// TIA Portal V16 export
// export: Created 2021-04-13T11:10:14.4344979Z, ExportSetting WithDefaults, DisplayName Totally Integrated Automation Portal, DisplayVersion V16, DisplayName TIA Portal Version Control Interface, DisplayVersion V16, DisplayName TIA Portal Openness, DisplayVersion V16, DisplayName STEP 7 Professional, DisplayVersion V16, DisplayName STEP 7 Safety, DisplayVersion V16, DisplayName WinCC Unified SCADA Engineering System, DisplayVersion V16
FUNCTION_BLOCK "modbus_SenecaConnectPort2"   // FB14, LAD
{ S7_Optimized_Access := 'TRUE' }
VERSION : 0.1
// stored: AutoNumber false, IsIECCheckEnabled false, IsRetainMemResEnabled false, MemoryReserve 100, SetENOAutomatically false, UDAEnableTagReadback false
   VAR_INPUT
      port : PORT;   // порт для подключения
      arrayAddressModbus : Array[0..12] of UInt;
      Offset_array_bits : SInt;
   END_VAR
   VAR_IN_OUT
      calibrateZero : Array[0..12] of Bool;
      taraZero : Array[0..12] of Bool;
      currentWeight : Array[0..12] of Real;
   END_VAR
   VAR
      MB_COMM_LOAD : MB_COMM_LOAD;
      MB_MASTER : MB_MASTER;
      Data_toMB_MASTER : Struct
         REQ : Bool;
         MB_ADDR : UInt;
         MODE : USInt;
         DATA_ADDR : UDInt;
         DATA_LEN : UInt;
         DONE : Bool;
         BUSY : Bool;
         ERROR : Bool;
      END_STRUCT;
      Seneca : Struct
         TON_changeStep : TON_TIME;
         TON_Start { S7_SetPoint := 'True'} : Bool;
         "Step" : SInt;
      END_STRUCT;
      tmpWeight : Array[0..12] of DWord;
      restartPort : Bool;   // перезагрузка Modbus
      needCalibrate : Bool;   // проверка на необходимость калибровки или тарирования
      testDone : Struct
         ton1 : TON_TIME;
         pulse_High : Bool;
         ton2 : TON_TIME;
         p_trig : Bool;
         ctu1 : CTU_INT;
      END_STRUCT;
   END_VAR
   VAR_TEMP
      index : DInt;
      tmpIndex : DInt;
      i : DInt;
   END_VAR
   // MB_COMM_LOAD.RETRIES := 1;
   VAR_TEMP   // added for the SCL form of the ladder/FBD networks
      _w1 : Bool;
   END_VAR
BEGIN

REGION Network 1: ИНИЦИАЛИЗИРУЕМ ПОРТ
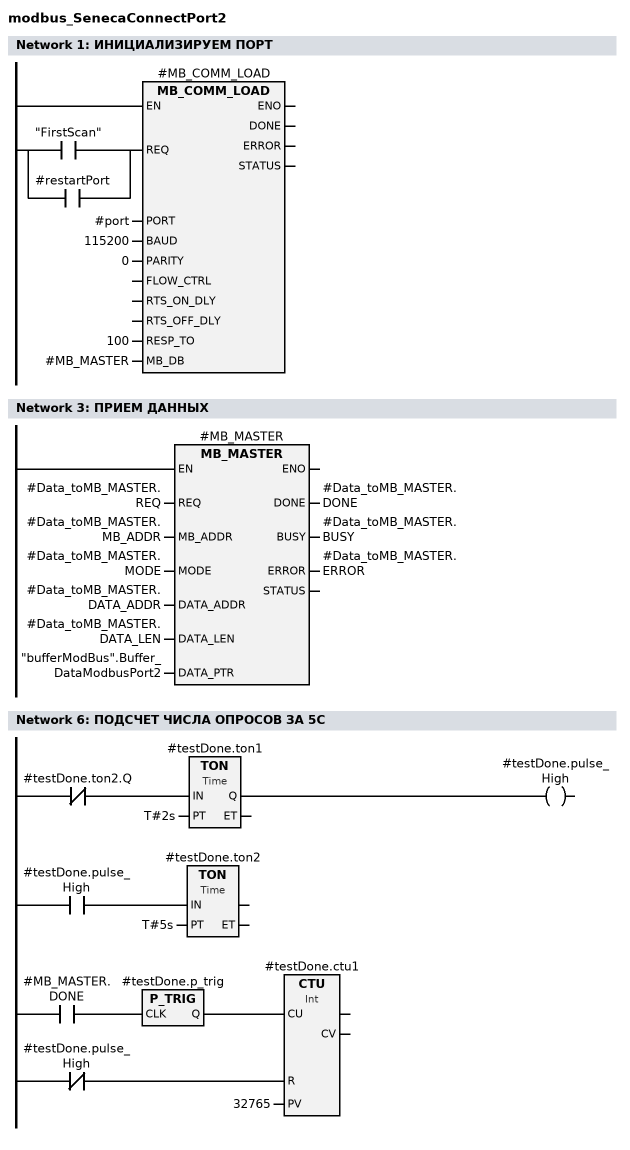
   RUNG wire#powerrail
      #MB_COMM_LOAD.MB_COMM_LOAD(REQ := wire#w1, PORT := #port, BAUD := 115200, PARITY := 0, FLOW_CTRL :=, RTS_ON_DLY :=, RTS_OFF_DLY :=, RESP_TO := 100, MB_DB := #MB_MASTER, DONE =>, ERROR =>, STATUS =>)
   END_RUNG
   RUNG wire#powerrail
      Contact( "FirstScan" )
   END_RUNG wire#w1
   RUNG wire#powerrail
      Contact( #restartPort )
   END_RUNG wire#w1
   // the same network as SCL:
   #MB_COMM_LOAD(REQ := "FirstScan" OR #restartPort,   // MB_COMM_LOAD
                 PORT := #port,
                 BAUD := 115200,
                 PARITY := 0,
                 RESP_TO := 100,
                 MB_DB := #MB_MASTER);
END_REGION

REGION Network 2 (SCL): ОБМЕН
   #Seneca.TON_changeStep(IN := #Seneca.TON_Start,
                          PT := t#50ms);

   CASE #Seneca.Step OF

       1: //ЧИТАЕМ ЗНАЧЕНИЕ ВЕСА С ПЕРВОГО МОДУЛЯ

           #index := 1 + #Offset_array_bits;//заполнять функцию будем через индекс чтобы меньше писать
           "rcvDataWeight"(ADDR_DEVICE := #arrayAddressModbus[#index],
                           Ton_changeStep := #Seneca.TON_changeStep.Q,
                           Ton_Start := #Seneca.TON_Start,
                           "Step" := #Seneca.Step,
                           MB_MASTER := #Data_toMB_MASTER);

       2://ЧИТАЕМ ЗНАЧЕНИЕ ВЕСА СО ВТОРОГО МОДУЛЯ
           #index := 2 + #Offset_array_bits;//заполнять функцию будем через индекс чтобы меньше писать
           "rcvDataWeight"(ADDR_DEVICE := #arrayAddressModbus[#index],
                           Ton_changeStep := #Seneca.TON_changeStep.Q,
                           Ton_Start := #Seneca.TON_Start,
                           "Step" := #Seneca.Step,
                           MB_MASTER := #Data_toMB_MASTER);

       7: // КАЛИБРОВКА 0 ДЛЯ ПЕРВОГО МОДУЛЯ и ТАРИРОВАНИЕ
           #i := 0;
           FOR #i := 1 TO 6 DO
               IF #calibrateZero[#i + #Offset_array_bits] OR #taraZero[#i + #Offset_array_bits] THEN
                   #needCalibrate := true;
                   EXIT;
               END_IF;
           END_FOR;

           IF #needCalibrate THEN
               #index := 1 + #Offset_array_bits;//заполнять функцию будем через индекс чтобы меньше писать
               IF #calibrateZero[#index] OR #taraZero[#index] THEN
                   "sndCALIBR&Tara"(ADDR_DEVICE := #arrayAddressModbus[#index],
                                    ton_changeStep := #Seneca.TON_changeStep.Q,
                                    MB_MASTER := #Data_toMB_MASTER,
                                    Ton_Start := #Seneca.TON_Start,
                                    Calibrate := #calibrateZero[#index],
                                    Buffer := "bufferModBus".Buffer_DataModbusPort2,
                                    "Step" := #Seneca.Step,
                                    Tara := #taraZero[#index]);
               ELSE
                   #Seneca.Step := #Seneca.Step + 1;
               END_IF;
           ELSE
               #Seneca.Step := 1;
           END_IF;

       8:// КАЛИБРОВКА 0 ДЛЯ ВТОРОГО МОДУЛЯ и ТАРИРОВАНИЕ
           #index := 2 + #Offset_array_bits;//заполнять функцию будем через индекс чтобы меньше писать
           IF #calibrateZero[#index] OR #taraZero[#index] THEN
               "sndCALIBR&Tara"(ADDR_DEVICE := #arrayAddressModbus[#index],
                                ton_changeStep := #Seneca.TON_changeStep.Q,
                                MB_MASTER := #Data_toMB_MASTER,
                                Ton_Start := #Seneca.TON_Start,
                                Calibrate := #calibrateZero[#index],
                                Buffer := "bufferModBus".Buffer_DataModbusPort2,
                                "Step" := #Seneca.Step,
                                Tara := #taraZero[#index]);
           ELSE
               #Seneca.Step := #Seneca.Step + 1;
           END_IF;

           //////////////////////////////////////////////////////////////////////////////////
           //////////////////////////////////////////////////////////////////////////////////
           //////////////////////////////////////////////////////////////////////////////////
           //////////////////////////////////////////////////////////////////////////////////
       3: //ЧИТАЕМ ЗНАЧЕНИЕ ВЕСА С ТРЕТЬЕГО МОДУЛЯ

           #index := 3 + #Offset_array_bits;//заполнять функцию будем через индекс чтобы меньше писать
           "rcvDataWeight"(ADDR_DEVICE := #arrayAddressModbus[#index],
                           Ton_changeStep := #Seneca.TON_changeStep.Q,
                           Ton_Start := #Seneca.TON_Start,
                           "Step" := #Seneca.Step,
                           MB_MASTER := #Data_toMB_MASTER);

       4://ЧИТАЕМ ЗНАЧЕНИЕ ВЕСА С ЧЕТВЕРТОГО МОДУЛЯ
           #index := 4 + #Offset_array_bits;//заполнять функцию будем через индекс чтобы меньше писать
           "rcvDataWeight"(ADDR_DEVICE := #arrayAddressModbus[#index],
                           Ton_changeStep := #Seneca.TON_changeStep.Q,
                           Ton_Start := #Seneca.TON_Start,
                           "Step" := #Seneca.Step,
                           MB_MASTER := #Data_toMB_MASTER);

       9:// КАЛИБРОВКА 0 ДЛЯ ТРЕТЬЕГО  МОДУЛЯ

           #index := 3 + #Offset_array_bits;//заполнять функцию будем через индекс чтобы меньше писать
           IF #calibrateZero[#index] OR #taraZero[#index] THEN
               "sndCALIBR&Tara"(ADDR_DEVICE := #arrayAddressModbus[#index],
                                ton_changeStep := #Seneca.TON_changeStep.Q,
                                MB_MASTER := #Data_toMB_MASTER,
                                Ton_Start := #Seneca.TON_Start,
                                Calibrate := #calibrateZero[#index],
                                Buffer := "bufferModBus".Buffer_DataModbusPort2,
                                "Step" := #Seneca.Step,
                                Tara := #taraZero[#index]);
           ELSE
               #Seneca.Step := #Seneca.Step + 1;
           END_IF;

       10://КАЛИБРОВКА 0 ДЛЯ ЧЕТВЕРТОГО МОДУЛЯ

           #index := 4 + #Offset_array_bits;//заполнять функцию будем через индекс чтобы меньше писать
           IF #calibrateZero[#index] OR #taraZero[#index] THEN
               "sndCALIBR&Tara"(ADDR_DEVICE := #arrayAddressModbus[#index],
                                ton_changeStep := #Seneca.TON_changeStep.Q,
                                MB_MASTER := #Data_toMB_MASTER,
                                Ton_Start := #Seneca.TON_Start,
                                Calibrate := #calibrateZero[#index],
                                Buffer := "bufferModBus".Buffer_DataModbusPort2,
                                "Step" := #Seneca.Step,
                                Tara := #taraZero[#index]);
           ELSE
               #Seneca.Step := #Seneca.Step + 1;
           END_IF;

           /////////////////////////////////////////////////////////////////////////////////
           ////////////////////////////////////////////////////////////////////////////////
           ////////////////////////////////////////////////////////////////////////////////
           ////////////////////////////////////////////////////////////////////////////////
       5: //ЧИТАЕМ ЗНАЧЕНИЕ ВЕСА С ПЯТОГО МОДУЛЯ
           #index := 5 + #Offset_array_bits;//заполнять функцию будем через индекс чтобы меньше писать
           "rcvDataWeight"(ADDR_DEVICE := #arrayAddressModbus[#index],
                           Ton_changeStep := #Seneca.TON_changeStep.Q,
                           Ton_Start := #Seneca.TON_Start,
                           "Step" := #Seneca.Step,
                           MB_MASTER := #Data_toMB_MASTER);

       6://ЧИТАЕМ ЗНАЧЕНИЕ ВЕСА С ШЕСТОГО МОДУЛЯ
           #index := 6 + #Offset_array_bits;//заполнять функцию будем через индекс чтобы меньше писать
           "rcvDataWeight"(ADDR_DEVICE := #arrayAddressModbus[#index],
                           Ton_changeStep := #Seneca.TON_changeStep.Q,
                           Ton_Start := #Seneca.TON_Start,
                           "Step" := #Seneca.Step,
                           MB_MASTER := #Data_toMB_MASTER);

       11:// КАЛИБРОВКА 0 ДЛЯ ПЯТОГО  МОДУЛЯ

           #index := 5 + #Offset_array_bits;//заполнять функцию будем через индекс чтобы меньше писать
           IF #calibrateZero[#index] OR #taraZero[#index] THEN
               "sndCALIBR&Tara"(ADDR_DEVICE := #arrayAddressModbus[#index],
                                ton_changeStep := #Seneca.TON_changeStep.Q,
                                MB_MASTER := #Data_toMB_MASTER,
                                Ton_Start := #Seneca.TON_Start,
                                Calibrate := #calibrateZero[#index],
                                Buffer := "bufferModBus".Buffer_DataModbusPort2,
                                "Step" := #Seneca.Step,
                                Tara := #taraZero[#index]);
           ELSE
               #Seneca.Step := #Seneca.Step + 1;
           END_IF;

       12:// КАЛИБРОВКА 0 ДЛЯ ШЕСТОГО МОДУЛЯ
           #index := 6 + #Offset_array_bits;//заполнять функцию будем через индекс чтобы меньше писать
           IF #calibrateZero[#index] OR #taraZero[#index] THEN
               "sndCALIBR&Tara"(ADDR_DEVICE := #arrayAddressModbus[#index],
                                ton_changeStep := #Seneca.TON_changeStep.Q,
                                MB_MASTER := #Data_toMB_MASTER,
                                Ton_Start := #Seneca.TON_Start,
                                Calibrate := #calibrateZero[#index],                            Buffer := "bufferModBus".Buffer_DataModbusPort2,
                                "Step" := #Seneca.Step,
                                Tara := #taraZero[#index]);
           ELSE
               #Seneca.Step := #Seneca.Step + 1;
           END_IF;
           #needCalibrate := false;
       ELSE
           #Seneca.Step := 1;
   END_CASE;
END_REGION

REGION Network 3: ПРИЕМ ДАННЫХ
   RUNG wire#powerrail
      #MB_MASTER.MB_MASTER(REQ := #Data_toMB_MASTER.REQ, MB_ADDR := #Data_toMB_MASTER.MB_ADDR, MODE := #Data_toMB_MASTER.MODE, DATA_ADDR := #Data_toMB_MASTER.DATA_ADDR, DATA_LEN := #Data_toMB_MASTER.DATA_LEN, DATA_PTR := "bufferModBus".Buffer_DataModbusPort2, DONE => #Data_toMB_MASTER.DONE, BUSY => #Data_toMB_MASTER.BUSY, ERROR => #Data_toMB_MASTER.ERROR, STATUS =>)
   END_RUNG
   // the same network as SCL:
   #MB_MASTER(REQ := #Data_toMB_MASTER.REQ,   // MB_MASTER
              MB_ADDR := #Data_toMB_MASTER.MB_ADDR,
              MODE := #Data_toMB_MASTER.MODE,
              DATA_ADDR := #Data_toMB_MASTER.DATA_ADDR,
              DATA_LEN := #Data_toMB_MASTER.DATA_LEN,
              DATA_PTR := "bufferModBus".Buffer_DataModbusPort2,
              DONE => #Data_toMB_MASTER.DONE,
              BUSY => #Data_toMB_MASTER.BUSY,
              ERROR => #Data_toMB_MASTER.ERROR);
END_REGION

REGION Network 4 (SCL): Авария опроса модуля
   #index := 0;
   CASE #Seneca.Step OF
       1,7:
           #index := 7;
       2,8:
           #index := 8;
       3,9:
           #index := 9;
       4,10:
           #index := 10;
       5,11:
           #index := 11;
       6,12:
           #index := 12;

   END_CASE;
   IF #Data_toMB_MASTER.ERROR THEN
       "hmi".alarmTest.bit[#index] := true;
   ELSIF #Data_toMB_MASTER.DONE THEN
       "hmi".alarmTest.bit[#index] := FALSE;
   END_IF;
END_REGION

REGION Network 5 (SCL)
   IF #Seneca.Step = 1 AND #Data_toMB_MASTER.DONE THEN
       #tmpIndex := 1 + #Offset_array_bits;
       #tmpWeight[#tmpIndex].%W0 := "bufferModBus".Buffer_DataModbusPort2[1];
       #tmpWeight[#tmpIndex].%W1 := "bufferModBus".Buffer_DataModbusPort2[0];
       #currentWeight[#tmpIndex] := DWORD_TO_REAL(#tmpWeight[#tmpIndex]);
       "bufferModBus".Buffer_DataModbusPort2[0] := 0;
       "bufferModBus".Buffer_DataModbusPort2[1] := 0;

   END_IF;

   IF #Seneca.Step = 2 AND #Data_toMB_MASTER.DONE THEN
       #tmpIndex := 2 + #Offset_array_bits;
       #tmpWeight[#tmpIndex].%W0 := "bufferModBus".Buffer_DataModbusPort2[1];
       #tmpWeight[#tmpIndex].%W1 := "bufferModBus".Buffer_DataModbusPort2[0];
       #currentWeight[#tmpIndex] := DWORD_TO_REAL(#tmpWeight[#tmpIndex]);
       "bufferModBus".Buffer_DataModbusPort2[0] := 0;
       "bufferModBus".Buffer_DataModbusPort2[1] := 0;
   END_IF;

   IF #Seneca.Step = 3 AND #Data_toMB_MASTER.DONE THEN
       #tmpIndex := 3 + #Offset_array_bits;
       #tmpWeight[#tmpIndex].%W0 := "bufferModBus".Buffer_DataModbusPort2[1];
       #tmpWeight[#tmpIndex].%W1 := "bufferModBus".Buffer_DataModbusPort2[0];
       #currentWeight[#tmpIndex] := DWORD_TO_REAL(#tmpWeight[#tmpIndex]);
       "bufferModBus".Buffer_DataModbusPort2[0] := 0;
       "bufferModBus".Buffer_DataModbusPort2[1] := 0;
   END_IF;

   IF #Seneca.Step = 4 AND #Data_toMB_MASTER.DONE THEN
       #tmpIndex := 4 + #Offset_array_bits;
       #tmpWeight[#tmpIndex].%W0 := "bufferModBus".Buffer_DataModbusPort2[1];
       #tmpWeight[#tmpIndex].%W1 := "bufferModBus".Buffer_DataModbusPort2[0];
       #currentWeight[#tmpIndex] := DWORD_TO_REAL(#tmpWeight[#tmpIndex]);
       "bufferModBus".Buffer_DataModbusPort2[0] := 0;
       "bufferModBus".Buffer_DataModbusPort2[1] := 0;
   END_IF;

   IF #Seneca.Step = 5 AND #Data_toMB_MASTER.DONE THEN
       #tmpIndex := 5 + #Offset_array_bits;
       #tmpWeight[#tmpIndex].%W0 := "bufferModBus".Buffer_DataModbusPort2[1];
       #tmpWeight[#tmpIndex].%W1 := "bufferModBus".Buffer_DataModbusPort2[0];
       #currentWeight[#tmpIndex] := DWORD_TO_REAL(#tmpWeight[#tmpIndex]);
       "bufferModBus".Buffer_DataModbusPort2[0] := 0;
       "bufferModBus".Buffer_DataModbusPort2[1] := 0;
   END_IF;

   IF #Seneca.Step = 6 AND #Data_toMB_MASTER.DONE THEN
       #tmpIndex := 6 + #Offset_array_bits;
       #tmpWeight[#tmpIndex].%W0 := "bufferModBus".Buffer_DataModbusPort2[1];
       #tmpWeight[#tmpIndex].%W1 := "bufferModBus".Buffer_DataModbusPort2[0];
       #currentWeight[#tmpIndex] := DWORD_TO_REAL(#tmpWeight[#tmpIndex]);
       "bufferModBus".Buffer_DataModbusPort2[0] := 0;
       "bufferModBus".Buffer_DataModbusPort2[1] := 0;
   END_IF;
END_REGION

REGION Network 6: ПОДСЧЕТ ЧИСЛА ОПРОСОВ ЗА 5С
   RUNG wire#powerrail
      I_Contact( #testDone.ton2.Q )
      { S7_Templates := "time_type := Time" } #testDone.ton1.TON(pt := T#2s, et =>)
      Coil( #testDone.pulse_High )
   END_RUNG
   RUNG wire#powerrail
      Contact( #testDone.pulse_High )
      { S7_Templates := "time_type := Time" } #testDone.ton2.TON(pt := T#5s, et =>)
   END_RUNG
   RUNG wire#powerrail
      Contact( #MB_MASTER.DONE )
      P_Trig( #testDone.p_trig )
      { S7_Templates := "value_type := Int" } #testDone.ctu1.CTU(r := wire#w1, pv := 32765, cv =>)
   END_RUNG
   RUNG wire#powerrail
      I_Contact( #testDone.pulse_High )
   END_RUNG wire#w1
   // the same network as SCL:
   #testDone.ton1.TON(IN := NOT #testDone.ton2.Q, PT := T#2s);
   #testDone.pulse_High := #testDone.ton1.Q;
   #testDone.ton2.TON(IN := #testDone.pulse_High, PT := T#5s);
   #_w1 := #MB_MASTER.DONE AND NOT #testDone.p_trig;   // rising edge
   #testDone.p_trig := #MB_MASTER.DONE;
   #testDone.ctu1.CTU(CU := #_w1, R := NOT #testDone.pulse_High, PV := 32765);
END_REGION
END_FUNCTION_BLOCK
